// TIA Portal V20 export
// export: Created 2025-12-01T14:57:09.5537032Z, ExportSetting None, DisplayName Totally Integrated Automation Portal, DisplayVersion V20 Update 3, DisplayName TIA Portal Openness, DisplayVersion V20 Update 3, DisplayName TIA Portal Version Control Interface, DisplayVersion V20 Update 3, DisplayName STEP 7 Professional, DisplayVersion V20 Update 3, DisplayName STEP 7 Safety, DisplayVersion V20 Update 2, DisplayName WinCC Basic/Comfort/Advanced, DisplayVersion V20 Update 3, DisplayName WinCC Professional, DisplayVersion V20 Update 3, DisplayName WinCC Unified, DisplayVersion V20 Update 3
FUNCTION "FC721_CrearUT_EnMesa" : Void   // FC721, LAD
TITLE = "CrearUT_EnMesa" - Crea una NUeva UT en la Mesa
{ S7_Optimized_Access := 'FALSE' }
AUTHOR : TRACKING
NAME : 20160108
VERSION : 3.2
// stored: AutoNumber false, SetENOAutomatically false
   VAR_INPUT
      McKey : UDInt;   // McKey de la UT
      MesaActual : UInt;   // Mesa Actual de la UT
   END_VAR
   VAR_OUTPUT
      NumeroUT : UInt;   // Nuemro de la UT Creada
   END_VAR
   VAR_TEMP
      Mesa : UInt;   // Mesa
      NumUT : UInt;   // Numero UT
      UTPrimera : UInt;   // UT Primera en la Mesa
      UTAnterior : UInt;   // UT Anterior en la Mesa
      UTSiguinte : UInt;   // UT Siguinte en la Mesa
      ColaMckey : UInt;   // Numnero de Cola de Ordenacion por Mckey
      TEMP_NumeroUT : UInt;
   END_VAR
BEGIN

NETWORK
TITLE = Inicilizar
// - Iniciliza numero de DB's
// - Iniciliza variables internas
////////////////////////////////////////////////////////////////////////////////
// Inicializa las variables
      L     0;  // Numero de UT Temporal
      T     #TEMP_NumeroUT;

      L     #MesaActual;  // Ver que mesa es
      T     #Mesa;



NETWORK
TITLE = Crear UT en Mesa -- Previo
////////////////////////////////////////////////////////////////////////////////
// Miro primero si hay alguna UT en la Cola de Mesa
      L     "DB810_ColasMesas".Colas[#Mesa].UT_PrimeraMesa;
      T     #UTPrimera;

      L     #UTPrimera;
      L     0;
      <>I;
      JC    HayUTs_EnColaMesa;  // Hay UT's en la Mesa
      JU    NoHayUTs_EnColaMesa;



NETWORK
TITLE = -- No Hay UT en la Cola de la Mesa
////////////////////////////////////////////////////////////////////////////////
////////////////////////////////////////////////////////////////////////////////
////////////////////////////////////////////////////////////////////////////////
// Mo hay UT's en la Cola de Mesa, Hay crear una
NoHayUTs_EnColaMesa:NOP   0;
      CALL  "FC723_InsertarUT_EnMesa"
      ( MesaActual := #MesaActual,
        NumeroUT   := #NumUT
      );

      L     0;  // NO hay Espacio para Mas UTs
      L     #NumUT;
      ==I;
      JC    Final_Funcion;


////////////////////////////////////////////////////////////////////////////////
// Ya tenemos la UT nueva, Y es la unica.
// Rellanar campos de la base de datos con lo basico
      L     #McKey;
      T     "DB812_UTs_Control".UT[#NumUT].Mckey;


      L     #MesaActual;
      L     "CTE_OffsetMesa";  // Mesa Actual Correcta
      +I;  // + Offset
      T     "DB812_UTs_Control".UT[#NumUT].MesaActual;


////////////////////////////////////////////////////////////////////////////////
// Relleno cual es la primera de la mesa
      L     #NumUT;
      T     "DB810_ColasMesas".Colas[#Mesa].UT_PrimeraMesa;

      JU    Final_EnColaMesa;



NETWORK
TITLE = -- Hay UT en la Cola de la Mesa
////////////////////////////////////////////////////////////////////////////////
////////////////////////////////////////////////////////////////////////////////
////////////////////////////////////////////////////////////////////////////////
// Hay UT's en la Cola de mesa
HayUTs_EnColaMesa:NOP   0;
      L     #UTPrimera;  // La UT Actual
      T     #NumUT;

      L     0;  // Inicio variables
      T     #UTAnterior;
      T     #UTSiguinte;


////////////////////////////////////////////////////////////////////////////////
// Empiezo a recorrer los datos de UT en la Mesa
BucleUT_EnMesa:NOP   0;

////////////////////////////////////////////////////////////////////////////////
//// CUIDADO CON ESTA CONDCION --- Se elimina
//Jose Antonio Alonso: Anulado 05/11/2015 para considerar que el MCkey 0 existe.
//porque llega el crea antes de enviar NUUT en movimientos dobles de la mesa

// "DB815_DatosUT".Datos_UTs[#NumUT].Mckey
//  L     0                           // Si es 0 es esta, la hemos creado ya
//   ==D
//   SPB MckeyCero_EnColaMesa
////////////////////////////////////////////////////////////////////////////////

      L     "DB812_UTs_Control".UT[#NumUT].UT_SiguienteMesa;
      L     0;  // Si es 0 es la ultima mesa, y hay crear una
      ==I;
      JC    FinalUT_EnColaMesa;

      L     "DB812_UTs_Control".UT[#NumUT].UT_SiguienteMesa;
      T     #NumUT;  // Mirar la siguiente de la Mesa
      JU    BucleUT_EnMesa;


////////////////////////////////////////////////////////////////////////////////
////////////////////////////////////////////////////////////////////////////////
// UT con Mckey 0, ya esta creada (NO SE UTILIZA ESTA PARTE)
MckeyCero_EnColaMesa:NOP   0;
      L     #McKey;
      T     "DB812_UTs_Control".UT[#NumUT].Mckey;

      L     #MesaActual;
      L     "CTE_OffsetMesa";  // Mesa Actual Correcta
      +I;  // + Offset
      T     "DB812_UTs_Control".UT[#NumUT].MesaActual;
      L     0;
      T     "DB812_UTs_Control".UT[#NumUT].MesaDestino;
      T     "DB812_UTs_Control".UT[#NumUT].MesaIntermedia;

      JU    Final_EnColaMesa;


////////////////////////////////////////////////////////////////////////////////
////////////////////////////////////////////////////////////////////////////////
// No hay UT con Mckey 0, hay que crear una al final de la Cola de Mesa
FinalUT_EnColaMesa:NOP   0;
      L     #NumUT;
      T     #UTAnterior;

      CALL  "FC723_InsertarUT_EnMesa"
      ( MesaActual := #MesaActual,
        NumeroUT   := #NumUT
      );

      L     0;
      L     #NumUT;
      ==I;
      JC    Final_Funcion;


////////////////////////////////////////////////////////////////////////////////
// Ya tenemos la UT nueva, Y es la unica.
// Rellanar campos de la base de datos con lo basico
      L     #UTAnterior;
      T     "DB812_UTs_Control".UT[#NumUT].UT_AnteriorMesa;

      L     #McKey;
      T     "DB812_UTs_Control".UT[#NumUT].Mckey;

      L     #MesaActual;
      L     "CTE_OffsetMesa";  // Mesa Actual Correcta
      +I;  // + Offset
      T     "DB812_UTs_Control".UT[#NumUT].MesaActual;


////////////////////////////////////////////////////////////////////////////////
// Relleno la anterior UT de la Mesa
      L     #NumUT;
      T     "DB812_UTs_Control".UT[#UTAnterior].UT_SiguienteMesa;

      JU    Final_EnColaMesa;



NETWORK
TITLE = -- Final
////////////////////////////////////////////////////////////////////////////////
////////////////////////////////////////////////////////////////////////////////
////////////////////////////////////////////////////////////////////////////////
Final_EnColaMesa:NOP   0;
      L     #NumUT;
      T     #TEMP_NumeroUT;


NETWORK
TITLE = Modificar la Ordenacion de Mckey -- Previo
////////////////////////////////////////////////////////////////////////////////
////////////////////////////////////////////////////////////////////////////////
////////////////////////////////////////////////////////////////////////////////
// Control del Mckey
      L     #McKey;  // Tiene Mckey
      L     0;
      ==D;
      JC    Final_Funcion;


////////////////////////////////////////////////////////////////////////////////
////////////////////////////////////////////////////////////////////////////////
////////////////////////////////////////////////////////////////////////////////
// Miro primero si hay alguna UT en la Cola de Mckey

      L     #McKey;
      L     10000;  // Son 10.000 las Colas de Mckey
      MOD;
      T     #ColaMckey;  // Numero de Cola de Mckey

      L     "DB811_ColasMckeys".Colas_Mckey[#ColaMckey].UT_PrimerMckey;
      T     #NumUT;

      L     #NumUT;
      L     0;
      ==I;  // No hay ninguna UT en la Cola ??????
      JC    NoHayUTs_EnColaMckey;
      JU    HayUTs_EnColaMckey;



NETWORK
TITLE = -- No Hay UT en la Cola de Ordenacion
////////////////////////////////////////////////////////////////////////////////
////////////////////////////////////////////////////////////////////////////////
////////////////////////////////////////////////////////////////////////////////
// Mo hay UT's en la Cola de Mckey
// ----- Es la primera UT de la Cola de Mckey
NoHayUTs_EnColaMckey:NOP   0;
      L     #TEMP_NumeroUT;
      T     "DB811_ColasMckeys".Colas_Mckey[#ColaMckey].UT_PrimerMckey;

      JU    Final_EnColaMcKey;



NETWORK
TITLE = -- Hay UT en la Cola de Ordenacion
////////////////////////////////////////////////////////////////////////////////
////////////////////////////////////////////////////////////////////////////////
////////////////////////////////////////////////////////////////////////////////
// Hay UT's en la Cola de Mckey
HayUTs_EnColaMckey:NOP   0;

//// CUIDADO CON ESTA CONDCION - AÑADIDO PARA INTEGRIDAD DE LA COLA DE MCKEYs
      L     #NumUT;  // Error en la Integredad de la Cola
      L     #TEMP_NumeroUT;  // Esta en la cola. IMPOSIBLE
      ==I;  // No hacer nada
      JC    Final_Funcion;


////////////////////////////////////////////////////////////////////////////////
// ---- No es la primera UT de la Cola de Mckey - Buscar cual es la ultima
BucleUT_EnColaMckey:NOP   0;
      L     #NumUT;
      T     #UTAnterior;

      L     "DB811_ColasMckeys".MckeyUT[#NumUT].UT_SiguienteMcKey;
      T     #NumUT;

      L     #NumUT;
      L     0;
      ==I;
      JC    FinalUT_EnColaMckey;  // Es la Ultima UT en la Cola ??????

//// CUIDADO CON ESTA CONDCION- AÑADIDO PARA INTEGRIDAD DE LA COLA DE MCKEYs
      L     #NumUT;  // Error en la Integredad de la Cola
      L     #TEMP_NumeroUT;  // Esta en la cola. IMPOSIBLE
      ==I;  // No hacer nada
      JC    Final_Funcion;

      JU    BucleUT_EnColaMckey;  // Continuar con la Cola de Mckey


////////////////////////////////////////////////////////////////////////////////
////////////////////////////////////////////////////////////////////////////////
////////////////////////////////////////////////////////////////////////////////
// Final de la Cola de Mckey
FinalUT_EnColaMckey:NOP   0;
      L     #TEMP_NumeroUT;  // Modificacion el la Ultima UT
      T     "DB811_ColasMckeys".MckeyUT[#UTAnterior].UT_SiguienteMcKey;

      L     #UTAnterior;  // Modificacion el la UT Creada
      T     "DB811_ColasMckeys".MckeyUT[#TEMP_NumeroUT].UT_AnteriorMckey;

      JU    Final_EnColaMcKey;



NETWORK
TITLE = --- Final
////////////////////////////////////////////////////////////////////////////////
////////////////////////////////////////////////////////////////////////////////
////////////////////////////////////////////////////////////////////////////////
// ----- No hay más final de la Ordenacion por Mckey
Final_EnColaMcKey:NOP   0;



NETWORK
TITLE = Devolucion de la Funcion
////////////////////////////////////////////////////////////////////////////////
////////////////////////////////////////////////////////////////////////////////
////////////////////////////////////////////////////////////////////////////////
Final_Funcion:NOP   0;
      L     #TEMP_NumeroUT;
      T     #NumeroUT;



END_FUNCTION
